(* IEC 61131-3 sources: IRIS-Project/LASAL CONTROL SOFTWARE/LasalProject_2025_09_12/Class/MoveTimer, 1 file *)

(* ---- MoveTimer.st ---- *)
(*!
<Class
	Name               = "MoveTimer"
	Revision           = "0.0"
	RealtimeTask       = "false"
	CyclicTask         = "true"
	DefCyclictime      = "100 ms"
	BackgroundTask     = "false"
	Sigmatek           = "false"
	OSInterface        = "false"
	HighPriority       = "false"
	Automatic          = "false"
	UpdateMode         = "Prescan"
	SharedCommandTable = "true"
	Objectsize         = "(530,120)">
	<Channels>
		<Server Name="ClassSvr" Visualized="false" Initialize="false" WriteProtected="true" Retentive="false"/>
		<Server Name="s_1_3_pelletMode" Visualized="false" Initialize="false" WriteProtected="false" Retentive="false"/>
		<Server Name="s_MovTimer1" Visualized="false" Initialize="false" WriteProtected="false" Retentive="false"/>
		<Server Name="s_MovTimer2" Visualized="false" Initialize="false" WriteProtected="false" Retentive="false"/>
		<Server Name="s_MovTimer3" Visualized="false" Initialize="false" WriteProtected="false" Retentive="false"/>
		<Server Name="s_Reset" Visualized="false" Initialize="false" WriteProtected="false" Retentive="false"/>
		<Server Name="s_StartStopTimer" Visualized="false" Initialize="false" WriteProtected="false" Retentive="false"/>
		<Client Name="c_SysDate" Required="true" Internal="false"/>
		<Client Name="c_SysTime" Required="true" Internal="false"/>
		<Client Name="c_timer" Required="true" Internal="false"/>
	</Channels>
</Class>
*)
MoveTimer : CLASS
  //Servers:
	ClassSvr 	: SvrChCmd_DINT;
	s_StartStopTimer 	: SvrCh_DINT;
	s_MovTimer1 	: SvrCh_DINT;
	s_MovTimer2 	: SvrCh_DINT;
	s_MovTimer3 	: SvrCh_DINT;
	s_Reset 	: SvrCh_DINT;
	s_1_3_pelletMode 	: SvrCh_DINT;
  //Clients:
	c_timer 	: CltChCmd_TimeDateLib;
	c_SysDate 	: CltCh_DINT;
	c_SysTime 	: CltCh_TIME_LSL;
  //Variables:
		v_hd_Date 	: HDINT;
		v_hd_Time_1_Start 	: HDINT;
		v_hd_Time_2_Start 	: HDINT;
		v_hd_Time_3_Start 	: HDINT;
		v_hd_Time_1_Stop 	: HDINT;
		v_hd_Time_2_Stop 	: HDINT;
		v_hd_Time_3_Stop 	: HDINT;
		v_day 	: UDINT;
		v_month 	: UDINT;
		v_year 	: UDINT;
		v_tot_minutes 	: DINT;
		case_Time 	: DINT;
		a 	: DINT;
		i 	: DINT;
		v_tot_seconds_1 	: DINT;
		v_tot_seconds_2 	: DINT;
		v_tot_seconds_3 	: DINT;
  //Functions:

	FUNCTION VIRTUAL GLOBAL Init;

	FUNCTION VIRTUAL GLOBAL CyWork
		VAR_INPUT
			EAX 	: UDINT;
		END_VAR
		VAR_OUTPUT
			state (EAX) 	: UDINT;
		END_VAR;
  //Tables:
	FUNCTION @STD
		VAR_OUTPUT
			ret_code	: CONFSTATES;
		END_VAR;
	FUNCTION GLOBAL TAB @CT_;
END_CLASS;

#pragma usingLtd TimeDateLib

FUNCTION VIRTUAL GLOBAL MoveTimer::CyWork
	VAR_INPUT
		EAX 	: UDINT;
	END_VAR
	VAR_OUTPUT
		state (EAX) 	: UDINT;
	END_VAR

  //READ ACTUAL TIME AND DATE FROM CLIENTS; shr for shift bits
  //v_hd_Date := c_SysDate.Read();
  //v_hd_Time_1_Start := c_SysTime.Read();

  ///v_seconds_1 := (v_hd_Time_1_Start AND 16#0000FF00) shr 8;
  //v_minutes_1 := (v_hd_Time_1_Start AND 16#00FF0000) shr 16;
  //v_hours_1   := (v_hd_Time_1_Start AND 16#FF000000) shr 24;

  //v_day     := (v_hd_Date AND 16#00000FF0) shr 4;
  //v_month   := (v_hd_Date AND 16#0000F000) shr 12;
  //v_year    := (v_hd_Date AND 16#FFFF0000) shr 16;

  if s_Reset.Read() then
     s_MovTimer1.Write(input:=0);
     s_MovTimer2.Write(input:=0);
     s_MovTimer3.Write(input:=0);
     case_Time:=0;
  end_if;

  case case_Time of

    0://START 1
      if s_StartStopTimer.Read() then
        v_hd_Time_1_Start := c_SysTime.Read();

        if s_1_3_pelletMode.Read()=1 then
          s_StartStopTimer.Write(input:=1);
          case_Time:=30;
        elsif s_1_3_pelletMode.Read()=0 then
          s_StartStopTimer.Write(input:=0);
          case_Time:=10;
        end_if;

      end_if;

    10://START 2

      if s_StartStopTimer.Read() then
        v_hd_Time_2_Start := c_SysTime.Read();
        s_StartStopTimer.Write(input:=0);
        case_Time:=20;
      end_if;

    20://START 3

       if s_StartStopTimer.Read() then
        v_hd_Time_3_Start := c_SysTime.Read();
        s_StartStopTimer.Write(input:=1);
        case_Time:=30;
      end_if;

    30://STOP 1

      if s_StartStopTimer.Read()=0 then
        v_hd_Time_1_Stop:= c_SysTime.Read();
        v_tot_seconds_1:=c_timer.TimeDiff(tim1:=v_hd_Time_1_Stop, tim2:=v_hd_Time_1_Start);
        s_StartStopTimer.Write(input:=1);
        case_Time:=35;
      end_if;
    35:
      s_MovTimer1.Write(input:=v_tot_seconds_1);
      if s_1_3_pelletMode.Read()=1 then
        case_Time:=60;
      elsif s_1_3_pelletMode.Read()=0 then
        case_Time:=40;
      end_if;

    40://STOP 2

      if s_StartStopTimer.Read()=0 then
        v_hd_Time_2_Stop:= c_SysTime.Read();
        v_tot_seconds_2 := c_timer.TimeDiff(tim1:=v_hd_Time_2_Stop, tim2:=v_hd_Time_2_Start);
        s_StartStopTimer.Write(input:=1);
        case_Time:=45;
      end_if;

    45:

      s_MovTimer2.Write(input:=v_tot_seconds_2);
      case_Time:=50;

    50://STOP 3

      if s_StartStopTimer.Read()=0 then
        v_hd_Time_3_Stop:= c_SysTime.Read();
        v_tot_seconds_3 := c_timer.TimeDiff(tim1:=v_hd_Time_3_Stop, tim2:=v_hd_Time_3_Start);
        s_StartStopTimer.Write(input:=1);
        case_Time:=55;
      end_if;

    55:
      s_MovTimer3.Write(input:=v_tot_seconds_3);
      case_Time:=60;

    60:

  end_case;

	state := READY;

END_FUNCTION

FUNCTION VIRTUAL GLOBAL MoveTimer::Init

END_FUNCTION
